FUNCTION_BLOCK TactTimeFB
VAR_INPUT
	bComfirmStart:BOOL;
	bOnOff:BOOL;



END_VAR
VAR_OUTPUT
	iTactTime:INT;
	iCurrentTimer:INT;


END_VAR
VAR
	StartCount: BOOL;
	ComfirmPulse: R_TRIG;
	clockPulse: BOOL;
	SecondPulse: CLOCK_PLS;
	AddPulse: R_TRIG;
	currentTimer: INT;
	delayOn: TON;
	PulseOffCount: R_TRIG;
	TimeReset: BOOL;
	DelayTimeron: TON;
	off: BOOL;
	DelayMove: TON;
	movetrig: R_TRIG;
END_VAR
VAR // added by the converter: edge detectors and wires of the graphical bodies
    _w1, _w3 : INT;
    _w2 : ANY;
END_VAR

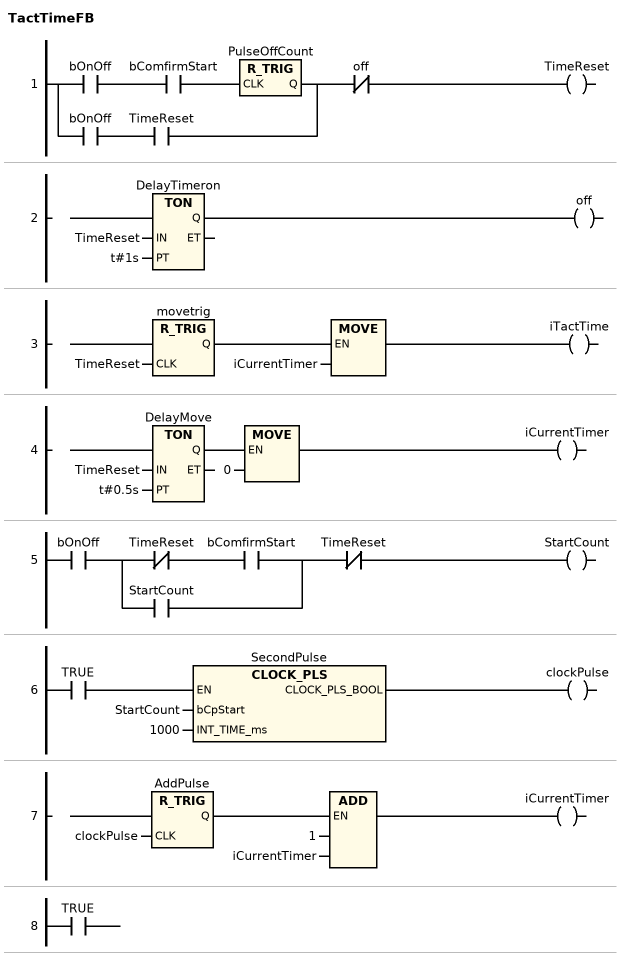
// NETWORK 1
PulseOffCount(CLK := bOnOff AND bComfirmStart); // R_TRIG
TimeReset := (PulseOffCount.Q OR bOnOff AND TimeReset) AND NOT off;

// NETWORK 2
DelayTimeron(IN := TimeReset, PT := t#1s); // TON
off := DelayTimeron.Q;

// NETWORK 3
movetrig(CLK := TimeReset); // R_TRIG
IF movetrig.Q THEN _w1 := iCurrentTimer; END_IF
iTactTime := _w1;

// NETWORK 4
DelayMove(IN := TimeReset, PT := t#0.5s); // TON
IF DelayMove.Q THEN _w2 := 0; END_IF
iCurrentTimer := _w2;

// NETWORK 5
StartCount := (bOnOff AND (NOT TimeReset AND bComfirmStart OR StartCount)) AND NOT TimeReset;

// NETWORK 6
SecondPulse(bCpStart := StartCount, INT_TIME_ms := 1000); // CLOCK_PLS
clockPulse := SecondPulse.CLOCK_PLS_BOOL;

// NETWORK 7
AddPulse(CLK := clockPulse); // R_TRIG
IF AddPulse.Q THEN _w3 := 1 + iCurrentTimer; END_IF
iCurrentTimer := _w3;

// NETWORK 8

END_FUNCTION_BLOCK

(* stored: Version 1.1.0.1, ProductVersion 3.1.4024.12
   POU TactTimeFB: Id {3b1e8642-8913-4d33-9c8a-1bcb076bf92e}, SpecialFunc None *)
